(* CODESYS project IoDrvSubModulesFixTest.project

Project tree, tasks and I/O mapping:
  Device : CODESYS Control Win V3, 3S - Smart Software Solutions GmbH, order no. 305021, version 3.5.9.0
    application Application
      libraries: Standard, * (System)
      task MainTask (cyclic, interval t#20ms, priority 1) calls PLC_PRG
      program PLC_PRG [ST]
    IoDrvSubModulesFix : IoDrvSubModulesFix, MyCompany, order no. 4711, version 3.5.9.0
      SubModuleForFixConnector : SubModuleForFixConnector, MyCompany, order no. abc, version 3.5.9.0
          output out1 : DWORD  // out1
          output out2 : DWORD  // out2
      SubModuleAsLocalModule : SubModuleAsLocalModule, MyCompany, order no. abc, version 3.5.9.0
          input  in1 : DWORD  // in1
          input  in2 : DWORD  // in2
*)

// Device/Application/PLC_PRG
PROGRAM PLC_PRG
VAR
END_VAR

in1;
in2;
out1 := out1 + 1;
out2;

END_PROGRAM
